// LS Electric XG5000 project: final_project
// PLC LSPLC

PROGRAM 00.Initialize (task: 스캔 프로그램)

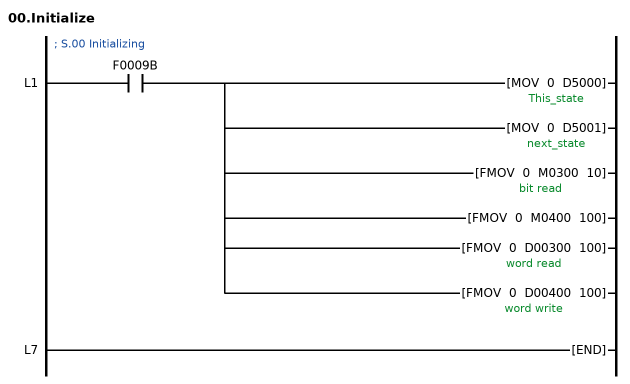
// S.00 Initializing
; L1
LOAD      F0009B
MOV       0 D5000	// This_state
MOV       0 D5001	// next_state
FMOV      0 M0300 10	// bit read
FMOV      0 M0400 100
FMOV      0 D00300 100	// word read
FMOV      0 D00400 100	// word write
; L7
END

PROGRAM InverterCom (task: 스캔 프로그램)

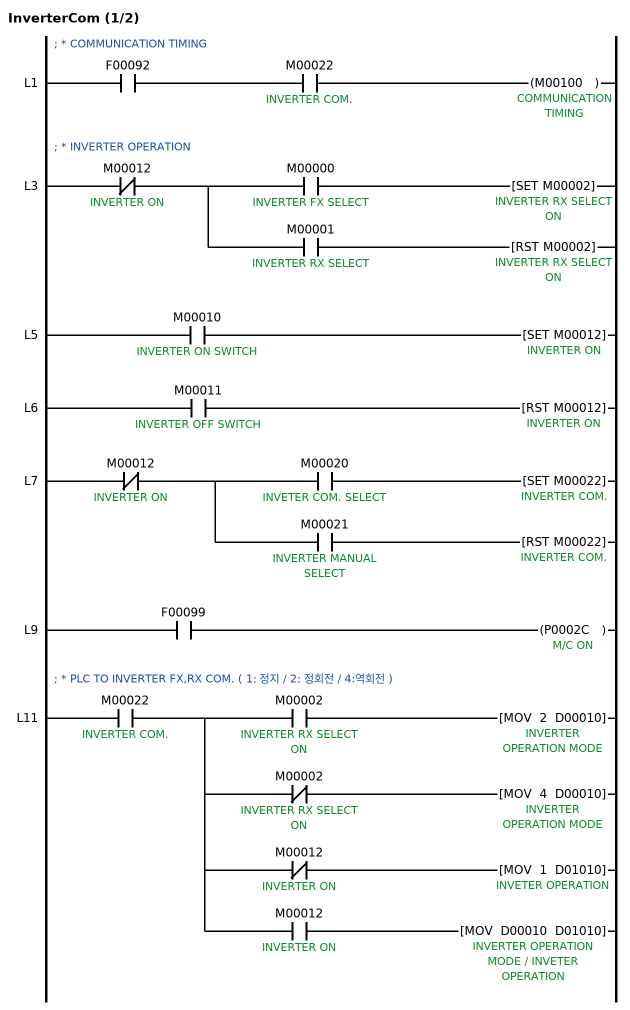
// * COMMUNICATION TIMING
; L1
LOAD      F00092
AND       M00022	// INVERTER COM.
OUT       M00100	// COMMUNICATION TIMING
// * INVERTER OPERATION
; L3
LOAD NOT  M00012	// INVERTER ON
MPUSH
AND       M00000	// INVERTER FX SELECT
SET       M00002	// INVERTER RX SELECT ON
MPOP
AND       M00001	// INVERTER RX SELECT
RST       M00002	// INVERTER RX SELECT ON
; L5
LOAD      M00010	// INVERTER ON SWITCH
SET       M00012	// INVERTER ON
; L6
LOAD      M00011	// INVERTER OFF SWITCH
RST       M00012	// INVERTER ON
; L7
LOAD NOT  M00012	// INVERTER ON
MPUSH
AND       M00020	// INVETER COM. SELECT
SET       M00022	// INVERTER COM.
MPOP
AND       M00021	// INVERTER MANUAL SELECT
RST       M00022	// INVERTER COM.
; L9
LOAD      F00099
OUT       P0002C	// M/C ON
// * PLC TO INVERTER FX,RX COM. ( 1: 정지 / 2: 정회전 / 4:역회전 )
; L11
LOAD      M00022	// INVERTER COM.
MPUSH
AND       M00002	// INVERTER RX SELECT ON
MOV       2 D00010	// INVERTER OPERATION MODE
MLOAD
AND NOT   M00002	// INVERTER RX SELECT ON
MOV       4 D00010	// INVERTER OPERATION MODE
MLOAD
AND NOT   M00012	// INVERTER ON
MOV       1 D01010	// INVETER OPERATION
MPOP
AND       M00012	// INVERTER ON
MOV       D00010 D01010	// INVERTER OPERATION MODE / INVETER OPERATION

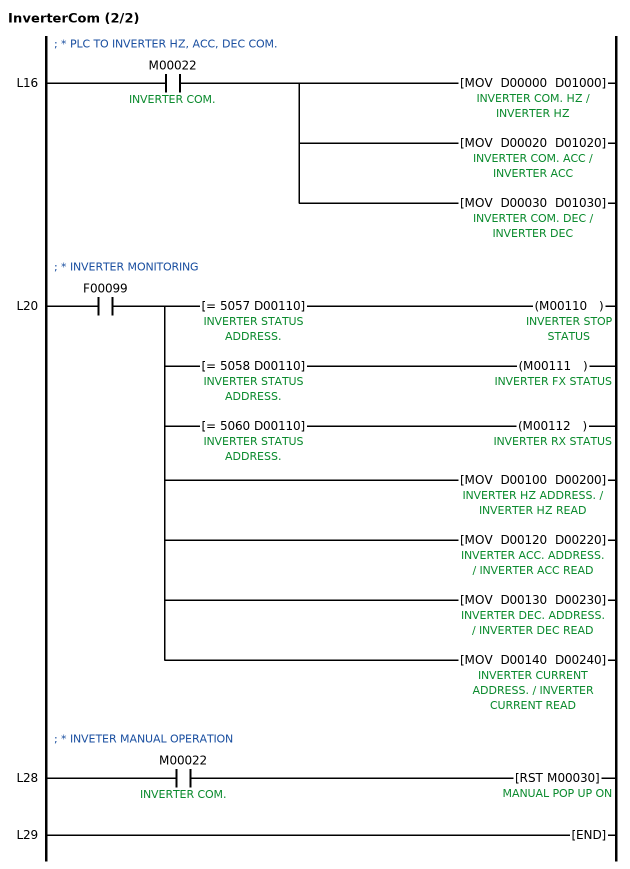
// * PLC TO INVERTER HZ, ACC, DEC COM.
; L16
LOAD      M00022	// INVERTER COM.
MOV       D00000 D01000	// INVERTER COM. HZ / INVERTER HZ
MOV       D00020 D01020	// INVERTER COM. ACC / INVERTER ACC
MOV       D00030 D01030	// INVERTER COM. DEC / INVERTER DEC
// * INVERTER MONITORING
; L20
LOAD      F00099
MPUSH
AND=      5057 D00110	// INVERTER STATUS ADDRESS.
OUT       M00110	// INVERTER STOP STATUS
MLOAD
AND=      5058 D00110	// INVERTER STATUS ADDRESS.
OUT       M00111	// INVERTER FX STATUS
MLOAD
AND=      5060 D00110	// INVERTER STATUS ADDRESS.
OUT       M00112	// INVERTER RX STATUS
MPOP
MOV       D00100 D00200	// INVERTER HZ ADDRESS. / INVERTER HZ READ
MOV       D00120 D00220	// INVERTER ACC. ADDRESS. / INVERTER ACC READ
MOV       D00130 D00230	// INVERTER DEC. ADDRESS. / INVERTER DEC READ
MOV       D00140 D00240	// INVERTER CURRENT ADDRESS. / INVERTER CURRENT READ
// * INVETER MANUAL OPERATION
; L28
LOAD      M00022	// INVERTER COM.
RST       M00030	// MANUAL POP UP ON
; L29
END

PROGRAM 10.Main (task: 스캔 프로그램)

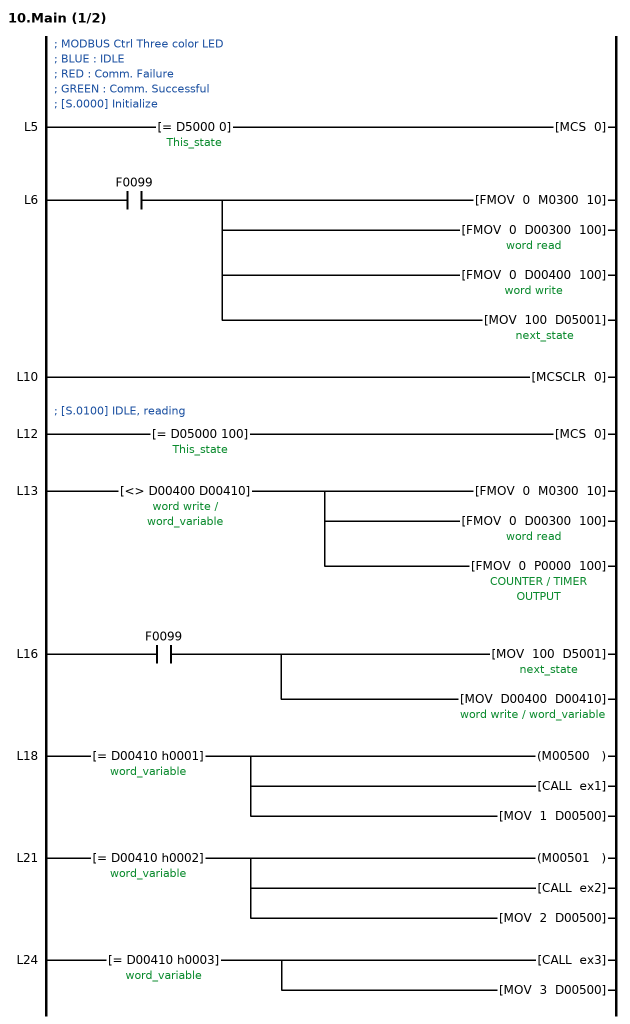
// MODBUS Ctrl Three color LED
// BLUE : IDLE
// RED : Comm. Failure
// GREEN : Comm. Successful
// [S.0000] Initialize
; L5
LOAD=     D5000 0	// This_state
MCS       0
; L6
LOAD      F0099
FMOV      0 M0300 10
FMOV      0 D00300 100	// word read
FMOV      0 D00400 100	// word write
MOV       100 D05001	// next_state
; L10
MCSCLR    0
// [S.0100] IDLE, reading
; L12
LOAD=     D05000 100	// This_state
MCS       0
; L13
LOAD<>    D00400 D00410	// word write / word_variable
FMOV      0 M0300 10
FMOV      0 D00300 100	// word read
FMOV      0 P0000 100	// COUNTER / TIMER OUTPUT
; L16
LOAD      F0099
MOV       100 D5001	// next_state
MOV       D00400 D00410	// word write / word_variable
; L18
LOAD=     D00410 h0001	// word_variable
OUT       M00500
CALL      ex1
MOV       1 D00500
; L21
LOAD=     D00410 h0002	// word_variable
OUT       M00501
CALL      ex2
MOV       2 D00500
; L24
LOAD=     D00410 h0003	// word_variable
CALL      ex3
MOV       3 D00500

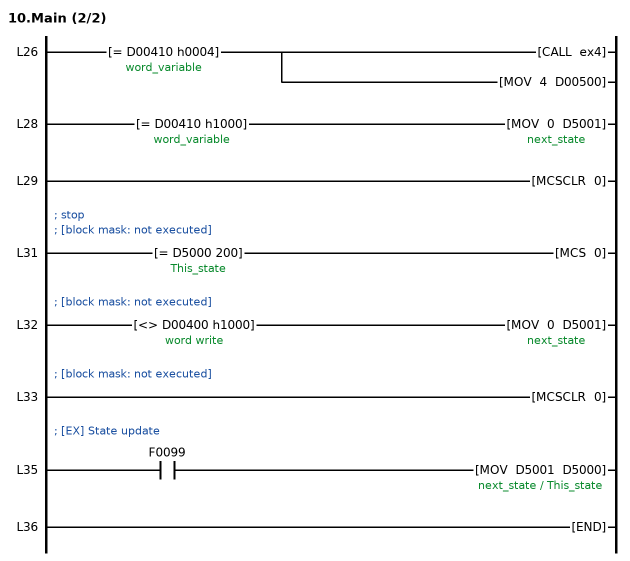
; L26
LOAD=     D00410 h0004	// word_variable
CALL      ex4
MOV       4 D00500
; L28
LOAD=     D00410 h1000	// word_variable
MOV       0 D5001	// next_state
; L29
MCSCLR    0
// stop
; L31 (block mask: not executed)
LOAD=     D5000 200	// This_state
MCS       0
; L32 (block mask: not executed)
LOAD<>    D00400 h1000	// word write
MOV       0 D5001	// next_state
; L33 (block mask: not executed)
MCSCLR    0
// [EX] State update
; L35
LOAD      F0099
MOV       D5001 D5000	// next_state / This_state
; L36
END

PROGRAM 20.IO_Ctrl (task: 스캔 프로그램)

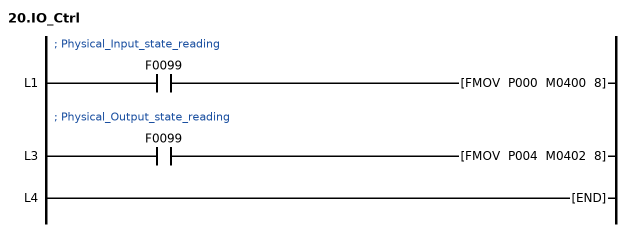
// Physical_Input_state_reading
; L1
LOAD      F0099
FMOV      P000 M0400 8
// Physical_Output_state_reading
; L3
LOAD      F0099
FMOV      P004 M0402 8
; L4
END

PROGRAM 99.DEF (task: 스캔 프로그램)

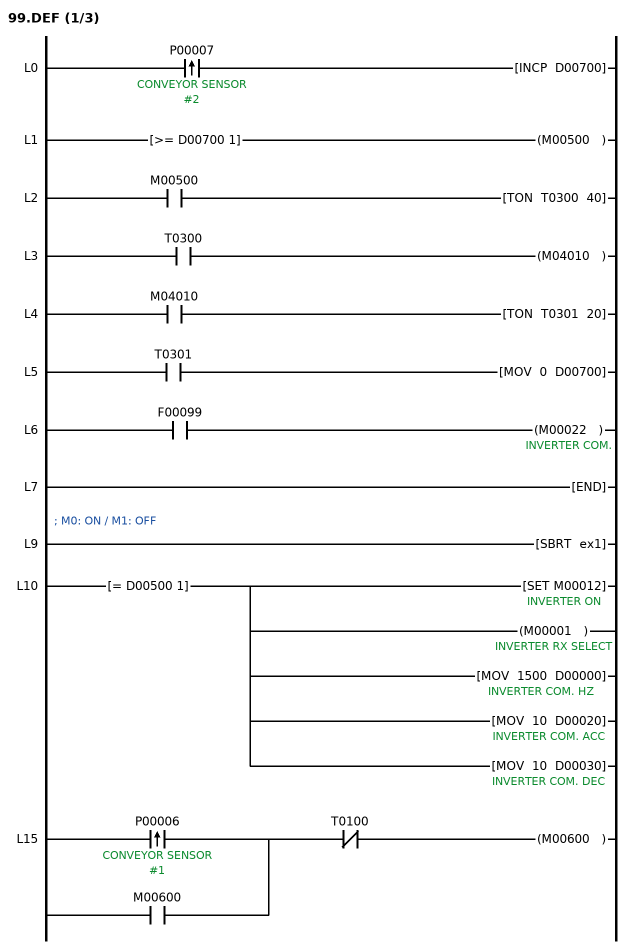
; L0
LOADP     P00007	// CONVEYOR SENSOR #2
INCP      D00700
; L1
LOAD>=    D00700 1
OUT       M00500
; L2
LOAD      M00500
TON       T0300 40
; L3
LOAD      T0300
OUT       M04010
; L4
LOAD      M04010
TON       T0301 20
; L5
LOAD      T0301
MOV       0 D00700
; L6
LOAD      F00099
OUT       M00022	// INVERTER COM.
; L7
END
// M0: ON / M1: OFF
; L9
SBRT      ex1
; L10
LOAD=     D00500 1
SET       M00012	// INVERTER ON
OUT       M00001	// INVERTER RX SELECT
MOV       1500 D00000	// INVERTER COM. HZ
MOV       10 D00020	// INVERTER COM. ACC
MOV       10 D00030	// INVERTER COM. DEC
; L15
LOADP     P00006	// CONVEYOR SENSOR #1
OR        M00600
AND NOT   T0100
OUT       M00600

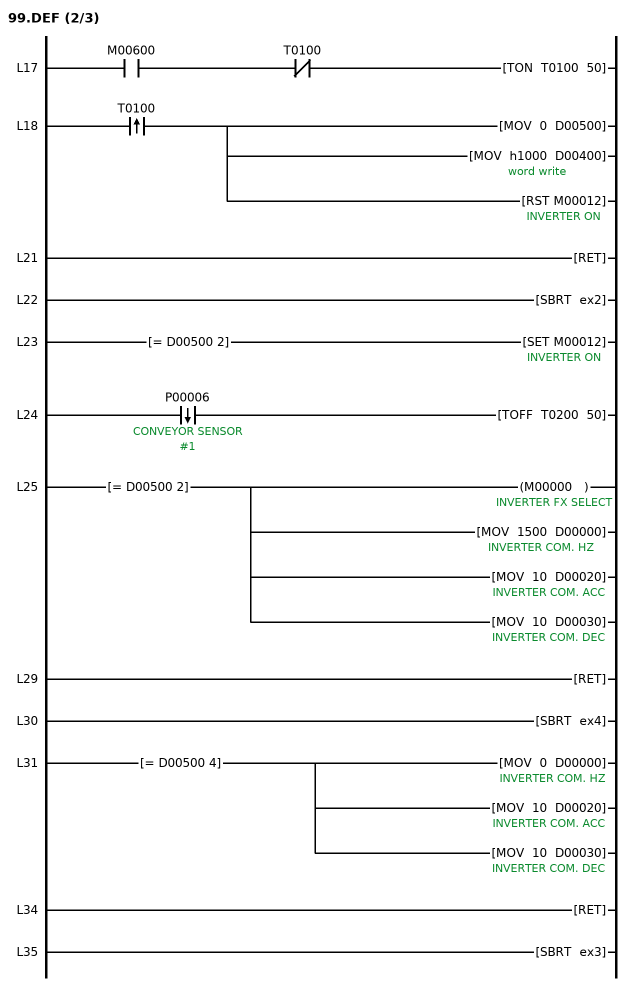
; L17
LOAD      M00600
AND NOT   T0100
TON       T0100 50
; L18
LOADP     T0100
MOV       0 D00500
MOV       h1000 D00400	// word write
RST       M00012	// INVERTER ON
; L21
RET
; L22
SBRT      ex2
; L23
LOAD=     D00500 2
SET       M00012	// INVERTER ON
; L24
LOADN     P00006	// CONVEYOR SENSOR #1
TOFF      T0200 50
; L25
LOAD=     D00500 2
OUT       M00000	// INVERTER FX SELECT
MOV       1500 D00000	// INVERTER COM. HZ
MOV       10 D00020	// INVERTER COM. ACC
MOV       10 D00030	// INVERTER COM. DEC
; L29
RET
; L30
SBRT      ex4
; L31
LOAD=     D00500 4
MOV       0 D00000	// INVERTER COM. HZ
MOV       10 D00020	// INVERTER COM. ACC
MOV       10 D00030	// INVERTER COM. DEC
; L34
RET
; L35
SBRT      ex3

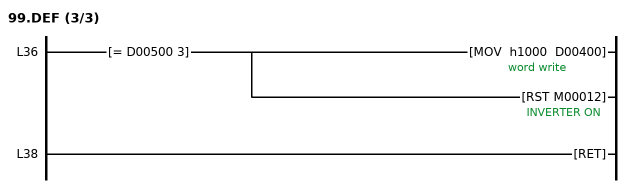
; L36
LOAD=     D00500 3
MOV       h1000 D00400	// word write
RST       M00012	// INVERTER ON
; L38
RET

VARIABLES AND COMMENTS (devices not used above)
M03000	BIT	1단 TOGGLE SWITCH
M03100	BIT	1단 TOGGLE SWITCH STATUS
M03001	BIT	2단 TOGGLE SWITCH ON
M03002	BIT	2단 TOGGLE SWITCH OFF
M03101	BIT	2단 TOGGLE SWITCH STATUS
M03003	BIT	1단 MOMENTARY SWITCH
M03005	BIT	2단 MOMENTARY SWITCH OFF
M03004	BIT	2단 MOMENTARY SWITCH ON
M03102	BIT	1단 MOMENTARY SWITCH STATUS
M03103	BIT	2단 MOMENTARY SWITCH STATUS
M02000	BIT	COUNT SELECT
M02001	BIT	TIMER SELECT
M02002	BIT	COUNTER INC
M02003	BIT	COUNTER DEC
M02004	BIT	TIMER INC
M02005	BIT	TIMER DEC
M02006	BIT	USED SENSOR
M02007	BIT	USED BUTTON
M02100	BIT	COUNTER / TIMER SELECT
M02101	BIT	COUNTER INC / DEC SELECT
M02102	BIT	TIMER INC / DEC SELECT
M02103	BIT	USED SENSOR / BUTTON SELECT
M02050	BIT	START SIGNAL
M02051	BIT	COUNT END SIGNAL
M02060	BIT	COUNTER USED SIGNAL
M02061	BIT	TIMER USED SIGNAL
M02053	BIT	TIMER END SIGNAL
M02054	BIT	TMON CHECK SIGNAL
M02055	BIT	TIMER RESET
M02052	BIT	COUNTER RESET
C0000	BIT/WORD	INC COUNTER
C0001	BIT/WORD	DEC COUNTER
D02000	WORD	COUNT
T0000	BIT/WORD	INC TIMER
T0001	BIT/WORD	DEC TIMER
D02010	WORD	TIME
D02020	WORD	TIMEX10
P00001	BIT	INVERTER OUTPUT
P00002	BIT	M/S ON STATUS
P00008	BIT	PUSH BUTTON ( TOGGLE )
P00009	BIT	PUSH BUTTON LIGHT
P0000A	BIT	PUSH BUTTON
P0000B	BIT	SELECT SWITCH - A
P0000C	BIT	SELECT SWITCH - B
P00020	BIT	COUNT PULSE
P00021	BIT	TIMER HOLD
P00022	BIT	RESET
P00024	BIT	RED LAMP ON
P00025	BIT	YELLOW LAMP ON
P00026	BIT	GREEN LAMP ON
P00028	BIT	INVERTER FX
P00029	BIT	INVERTER RX